FUNCTION_BLOCK T_BaseAlarmsClearAlarmIfRaisedCleared EXTENDS T_UnitTestBase
VAR
	baseAlarms : T_BaseAlarms;
END_VAR

//Arrange
baseAlarms.RaiseAlarmWithStringParameters(E_BaseAlarms.ComponentError, '','','');

//Act
baseAlarms.ClearAlarmIfRaised(E_BaseAlarms.ComponentError, resetConfirmation := FALSE);

//Assert
Assertion.AssertEquals_BOOL(Expected:= FALSE, Actual := TRUE, 
						VariableName:= 'baseAlarms.ClearAlarmIfRaised(E_BaseAlarms.ComponentError, resetConfirmation := FALSE);' );
TestFinished();

END_FUNCTION_BLOCK

(* stored: Version 1.1.0.1, ProductVersion 3.1.4024.12
   POU T_BaseAlarmsClearAlarmIfRaisedCleared: Id {720ccca1-1231-4aaa-bd2b-90b344432fcc}, SpecialFunc None *)
